TYPE ST_AxisGroupFlag :
STRUCT
	iError : INT;
	iDisabled : INT;
	iState : INT;
	bErrorFlag : BOOL;
	bDisabledFlag : BOOL;
	iNumberOfAxisInError : INT;
	iNumberOfAxisDisabled : INT;
END_STRUCT
END_TYPE

(* stored: Version 1.1.0.1, ProductVersion 3.1.4024.11
   DUT ST_AxisGroupFlag: Id {4d5f5484-dd5b-461a-8e7e-33d95add3131} *)
